Fanuc KAREL source: CONVERT_PARAMS.KL

PROGRAM CONVERT_PARAMS
%STACKSIZE = 4000
%NOLOCKGROUP
%NOPAUSE=ERROR+COMMAND+TPENABLE
%ENVIRONMENT uif
%ENVIRONMENT sysdef
%ENVIRONMENT memo
%ENVIRONMENT kclop
%ENVIRONMENT bynam
%ENVIRONMENT fdev
%ENVIRONMENT flbt
%ENVIRONMENT regope
%INCLUDE klevccdf
%INCLUDE klevkeys
%INCLUDE klevkmsk

CONST
    RIFTEK_DEFAULT_COMMAND = 128
-------------------------------------------------------------------------------------------------------
------------------------------------PARAMETERS CONVERSION----------------------------------------------
--CONVERT DECIMAL PARAMETER CODE TO RIFTEK HEXADECIMAL BYTE ARRAY WITH LENGTH = param_size * 2
--1 BYTE PARAMETER --> PARAMETER CODE -- 5 -->  5 * 16 ^ 1 -->  [5, 0] --> [133, 128],
--2 BYTE PARAMETER --> PARAMETER FIRST CODE -- 0A -->[0A, 0B] --> [10, 11] --> [138, 128, 139, 128]
ROUTINE CNV_DECIMAL_PARAM_TO_BYTE_ARRAY(param : INTEGER; param_size : INTEGER) : ARRAY OF BYTE
VAR
    byte_parameter : ARRAY[20] OF BYTE
    comparation_value : REAL
    shift_value : REAL
    index : INTEGER
BEGIN
    comparation_value = 15
    shift_value = 1
    FOR INDEX = 1 TO param_size * 2 DO
        byte_parameter[INDEX] = RIFTEK_DEFAULT_COMMAND +TRUNC((param AND TRUNC(comparation_value)) / shift_value)
        comparation_value = comparation_value * EXP(4 * LN(2))
        shift_value = shift_value * EXP(4 * LN(2))
    ENDFOR
    RETURN (byte_parameter)
END CNV_DECIMAL_PARAM_TO_BYTE_ARRAY

--CONVERT DECIMAL PARAMETER VALUE TO RIFTEK HEXADECIMAL BYTE ARRAY WITH LENGTH = param_size * 2
--1 BYTE PARAMETER --> PARAMETER VALUE -- 5 -->  5 * 16 ^ 1 -->  [5, 0] --> [133, 128],
--2 BYTE PARAMETER --> PARAMETER VALUE -- 3200 --> 0000 1100 1000 0000 --> [12(0000 11000), 128(1000 0000)] --> [0, 12, 8, 0] --> [128, 140, 136, 128]
ROUTINE CNV_DECIMAL_PARAM_CODE_TO_BYTE_ARRAY(param_code : INTEGER; param_size : INTEGER) : ARRAY OF BYTE
VAR
    byte_parameter : ARRAY[20] OF BYTE
    comparation_value : REAL
    shift_value : REAL
    out_index : INTEGER
    in_index : INTEGER
BEGIN
    FOR out_index = 1 TO param_size * 2 DO
        comparation_value = 15
        shift_value = 1
        FOR in_index = 0 TO 1 DO
            byte_parameter[out_index + in_index] = RIFTEK_DEFAULT_COMMAND + TRUNC((param_code AND TRUNC(comparation_value)) / shift_value)
            comparation_value = comparation_value * EXP(4 * LN(2))
            shift_value = shift_value * EXP(4 * LN(2))
        ENDFOR
        out_index = out_index + 1
        param_code = param_code + 1
    ENDFOR
    RETURN (byte_parameter)
END CNV_DECIMAL_PARAM_CODE_TO_BYTE_ARRAY

--CONVERT RIFTEK RESPONSE BYTE MESSAGE TO INTEGER PARAMETER
--[128, 140, 136, 128] --> [0, 12, 8, 0] --> [12(0000 11000), 128(1000 0000)] --> 3200
ROUTINE READ_PARAMETER_FROM_BYTE_ARRAY(response : ARRAY OF BYTE; start_byte_number : INTEGER; bytes_count : INTEGER) : INTEGER
VAR
    param_value : REAL
    multiplier : INTEGER
    power : INTEGER
    index : INTEGER
BEGIN
    param_value = 0
    multiplier = bytes_count * 2 - 1
    FOR INDEX = start_byte_number + bytes_count * 2 - 1 DOWNTO start_byte_number DO
        power = multiplier * 4
        param_value = param_value + ((response[index] AND 15) * EXP(power * LN(2)))
        multiplier = multiplier - 1
    ENDFOR
    RETURN (TRUNC(param_value))
END READ_PARAMETER_FROM_BYTE_ARRAY
------------------------------------PARAMETERS CONVERSION----------------------------------------------
-------------------------------------------------------------------------------------------------------
BEGIN
END CONVERT_PARAMS
